// TwinCAT 3 PLC project PLC_FIS
// ProgramVersion: 3.1.4024.12
// libraries:
//   Tc2_Standard, * (Beckhoff Automation GmbH)
//   Tc2_System, * (Beckhoff Automation GmbH)
//   Tc3_Module, * (Beckhoff Automation GmbH)
// project tree:
//   DUTs/ eAndMethod.TcDUT, eDeffuzyMethod.TcDUT (not stored), eOrMethod.TcDUT (not stored), eTest.TcDUT, MAMFIS.TcDUT, FIS_RULES.TcDUT, FIS_VAR.TcDUT, FIS_VAR_1.TcDUT (not stored), MF_INDEX.TcDUT, MF_SHAPE.TcDUT, MEMBERSHIP_FUNCTION.TcDUT (not stored)
//   GVLs/ gvlFIS_Constants.TcGVL
//   Old/ fbFuzzyAnd.TcPOU, fCentroidOld.TcPOU, fIntegrateMf.TcPOU, fIntExtFun.TcPOU, fis_cfc.TcPOU, fLinInterpol.TcPOU, LINEAR_LUT.TcPOU, LINEAR_LUT_old.TcPOU, mySumFb.TcPOU, testReferenceToFB.TcPOU
//   OOP/ FB_FIS_oop.TcPOU, FuzzyInferenceSystem.TcIO, OOP_MAIN.TcPOU
//   / PlcTask.TcTTO (not stored)
//   POP/Deffuzzification/ fCentroid.TcPOU (not stored)
//   POP/ FB_AGGREGATION.TcPOU (not stored), FB_IMPLICATION.TcPOU (not stored), FIS_pgr.TcPOU, MAIN.TcPOU
//   POP/Fuzzification/ fMembershipDegree.TcPOU, fMembershipDegreeArray.TcPOU
//   POP/Fuzzification/Membership Functions/ MF_Gaussian.TcPOU, MF_L.TcPOU, MF_R.TcPOU, MF_S.TcPOU (not stored), MF_Sigmoidal.TcPOU, MF_Singleton.TcPOU, MF_Trapezoidal.TcPOU (not stored), MF_Triangular.TcPOU, MF_Z.TcPOU
//   POP/FuzzyOperations/ fuzzyset.TcPOU, FuzzyAND_array.TcPOU (not stored), fuzzyAND.TcPOU, FuzzyNOT.TcPOU, FuzzyOR_array.TcPOU (not stored), FuzzyOR.TcPOU
//   POP/FuzzyOperations/T-Norms/ TN_min.TcPOU (not stored), TN_prod.TcPOU
//   POP/Test/ Test_fbFis.TcPOU (not stored)
//   POP/_FuzzyInferenceSystem/ FB_FIS_MAMDANI.TcPOU

// ---- DUTs/eAndMethod.TcDUT
//{attribute 'qualified_only'}
{attribute 'strict'}
TYPE eAndMethod :
(
	Minimum,
	Product
);
END_TYPE

// ---- DUTs/eTest.TcDUT
{attribute 'qualified_only'}
{attribute 'strict'}
TYPE eTest :
(
	enum_member := 0
);
END_TYPE

// ---- DUTs/MAMFIS.TcDUT
TYPE MAMFIS :
	STRUCT
		Name:STRING;
		Rules:ARRAY[1..NumOfFisRules]OF FIS_RULES;
		AndMethod:eAndMethod;
		OrMethod:eOrMethod;
		ImplicationMethod:eAndMethod; 
		AggregationMethod:eOrMethod;
		DefuzzificationMethod:eDeffuzyMethod;
		Inputs:ARRAY[1..NumOfFISInputs]OF FIS_VAR;
		MD:ARRAY[1..NumOfFISInputs,1..MFmax]OF REAL;//MD
		Outputs:ARRAY[1..NumOfFISOutputs]OF FIS_VAR;
	END_STRUCT
END_TYPE

// ---- DUTs/FIS_RULES.TcDUT
TYPE FIS_RULES :
STRUCT
	Antecedent: REAL;
	Consequents:ARRAY[1..NumOfFISOutputs]OF MF_INDEX;
END_STRUCT
END_TYPE

// ---- DUTs/FIS_VAR.TcDUT
TYPE FIS_VAR :
STRUCT
	CrispValue:REAL;
	Name:STRING;
	Range:ARRAY[1..2] OF REAL;
	NumberOfMF:INT;
	MF:ARRAY [1..MFmax]OF MEMBERSHIP_FUNCTION;//MF

END_STRUCT
END_TYPE

// ---- DUTs/MF_INDEX.TcDUT
TYPE
	MF_INDEX : INT;
END_TYPE

// ---- DUTs/MF_SHAPE.TcDUT
{attribute 'qualified_only'}
{attribute 'strict'}
TYPE MF_SHAPE :
(
	Gaussian,
	Lshaped,
	Rshaped,
	Sshaped,
	Sigmoidal,
	Singleton,
	Trapeziodal,
	Triangular,
	Zshaped
);
END_TYPE

// ---- GVLs/gvlFIS_Constants.TcGVL
{attribute 'global'}
VAR_GLOBAL CONSTANT
	NumOfFISInputs:INT :=	2;
	NumOfFISOutputs:INT := 	1;
	MFmax:INT := 			3;//maximum of MF per variable
	NumOfFisRules:INT := 	3;
	
	//inputs
	 	Error:INT:=1;
	 	Speed:INT:=2;
		
	//outputs
	 	power:INT:=1;
		
	//INPUT MEMBERSHIP FUNCTIONS
		None:INT := 	 1;
		Little:INT := 	 2;	
		Big:INT := 	 3;		
		//Negative:INT := 1;
		//Null:INT :=	 2;
		//Positive:INT := 3;
		
	//OUTPUT MEMBERSHIP FUNCTIONS
		Low:INT := 1;
		Medium:INT :=	 2;
		High:INT := 3;
END_VAR

// ---- OOP/FuzzyInferenceSystem.TcIO
INTERFACE FuzzyInferenceSystem

METHOD Defuzzification :REAL;
VAR_INPUT
END_VAR
END_METHOD

METHOD Fuzzyfication 
VAR_INPUT
END_VAR
END_METHOD

END_INTERFACE

// ---- Old/fbFuzzyAnd.TcPOU
FUNCTION_BLOCK fbFuzzyAnd
VAR_INPUT
END_VAR
VAR_OUTPUT
END_VAR
VAR
END_VAR

END_FUNCTION_BLOCK

// ---- Old/fCentroidOld.TcPOU
FUNCTION fCentroidOld : REAL
VAR_INPUT
	Range:ARRAY[1..2] OF REAL;
	MF:MEMBERSHIP_FUNCTION;
	Resolution:DINT;
END_VAR
VAR
	i:DINT;
	Xi,MDi,Step:REAL;
	Dividend:REAL:=0;//sum(MD(Xi))
 	Divisor:REAL:=0;//sum(Xi*MD(Xi))
END_VAR

(*
centroid=   sum(MD(Xi))  dividend
		  ==============
		  sum(Xi*MD(Xi)) divisor
*)
Step:=Range[2]-Range[1];
IF Resolution<>0 THEN
	FOR i := 1 TO resolution DO
		Xi := DINT_TO_REAL(i)*Step/Resolution;
		MDi := fMembershipDegree(Xi,MF);
		Dividend := Dividend + MDi;
		Divisor :=Divisor+(Mdi*Xi);
	END_FOR
	IF Divisor<>0 THEN
		fCentroidOld := Dividend/Divisor;
	ELSE
		fCentroidOld:=0;
	END_IF
ELSE fCentroidOld:=666;	
END_IF

END_FUNCTION

// ---- POP/Fuzzification/fMembershipDegree.TcPOU
FUNCTION fMembershipDegree : real
VAR_INPUT
	CrispInput: REAL;
	MF:MEMBERSHIP_FUNCTION;
END_VAR

VAR_OUTPUT
	error: BOOL;
END_VAR

CASE MF.Shape OF
	MF_SHAPE.Gaussian://********
		fMembershipDegree:=
			MF_Gaussian(
				x:= CrispInput,
				c:= MF.Points[1],
				d:= MF.Points[2],
				Error=>error);
	MF_SHAPE.Lshaped://********
		fMembershipDegree:=
			MF_L(
				x:= CrispInput,
				a:= MF.Points[1],
				b:= MF.Points[2],
				Error=>error);

	MF_SHAPE.rshaped://********
		fMembershipDegree:=
			MF_R(
				x:= CrispInput,
				c:= MF.Points[1],
				d:= MF.Points[2],
				Error=>error);
	
	MF_SHAPE.Sshaped://********
		fMembershipDegree:=
			MF_S(
				x:= CrispInput,
				a:= MF.Points[1],
				b:= MF.Points[2],
				Error=>error);

	MF_SHAPE.Sigmoidal://********
		fMembershipDegree:=
			MF_Gaussian(
				x:= CrispInput,
				d:= MF.Points[1],
				c:= MF.Points[2],
				Error=>error);
							
	MF_SHAPE.Singleton://********
		fMembershipDegree:=
			MF_Singleton(
				x:= CrispInput,
				a:= MF.Points[1]);
				
	MF_SHAPE.Trapeziodal://********
		fMembershipDegree:=
			MF_Trapezoidal(
				x:= CrispInput,
				a:= MF.Points[1],
				b:= MF.Points[2],
				c:= MF.Points[3],
				d:= MF.Points[3],
				Error=>error);
	
	MF_SHAPE.Triangular://********	
		fMembershipDegree:=
			MF_Triangular(
				x:= CrispInput,
				a:= MF.Points[1],
				m:= MF.Points[2],
				b:= MF.Points[3],
				error=>error);
				
	MF_SHAPE.Zshaped://********
		fMembershipDegree:=
			MF_R(
				x:= CrispInput,
				c:= MF.Points[1],
				d:= MF.Points[2],
				Error=>error);
	ELSE
		error:=TRUE;
	END_CASE;

END_FUNCTION

// ---- POP/Fuzzification/Membership Functions/MF_Gaussian.TcPOU
FUNCTION MF_Gaussian : real
VAR_INPUT
	x,d,c:REAL;(*Membership function parameters,
specified as the vector [d c], where σ is the 
standard deviation AND c is the mean.*)
END_VAR
VAR_OUTPUT
	Error:BOOL;
END_VAR

IF NOT(d=0) THEN
	MF_Gaussian := LREAL_TO_REAL(EXP(-EXPT((x-c),2)/EXPT(2*d,2)));
ELSE
	Error:=TRUE;
END_IF

END_FUNCTION

// ---- POP/Fuzzification/Membership Functions/MF_L.TcPOU
FUNCTION MF_L : real
VAR_INPUT
	x,a,b:REAL;(*a defines the foot of the membership function, AND b defines its shoulder.*)

END_VAR
VAR_OUTPUT
	Error:BOOL;
END_VAR

IF NOT(a=b) AND (a<b) THEN
	IF x<a THEN
		MF_L:=0;
	ELSIF a<=x AND x<=b THEN
		MF_L:=(x-a)/(b-a);
	ELSIF  x>b THEN
		MF_L:=1;
	END_IF
ELSE
	Error:=TRUE;		
END_IF

END_FUNCTION

// ---- POP/Fuzzification/Membership Functions/MF_R.TcPOU
 FUNCTION MF_R : real
VAR_INPUT
	x,d,c:REAL;(*a defines the foot of the membership function, AND b defines its shoulder.*)

END_VAR
VAR_OUTPUT
	Error:BOOL;
END_VAR

IF NOT(c=d) AND (c<d) THEN
	IF x>d THEN
		MF_R:=0;
	ELSIF c<=x AND x<=d THEN
		MF_R:=(d-x)/(d-c);
	ELSIF  x<c THEN
		MF_R:=1;
	END_IF
ELSE
	Error:=TRUE;		
END_IF

END_FUNCTION

// ---- POP/Fuzzification/Membership Functions/MF_Singleton.TcPOU
FUNCTION MF_Singleton : real
VAR_INPUT
	x,a:REAL;
END_VAR
VAR
END_VAR

IF x=a then
	MF_Singleton:=1;
ELSE
	MF_Singleton:=0;
END_IF

END_FUNCTION

// ---- POP/Fuzzification/Membership Functions/MF_Triangular.TcPOU
FUNCTION MF_Triangular : real
VAR_INPUT
	x,a,m,b:REAL;
END_VAR
VAR_OUTPUT
	error: BOOL;
END_VAR

// a < m < b
IF (a<m) AND (m<b) THEN
	IF x<=a OR x>=b THEN
		MF_Triangular:=0;
	ELSIF a<x AND x<m THEN
		MF_Triangular:=(x-a)/(m-a);
	ELSIF m<=x AND x<=b THEN
		MF_Triangular:=(b-x)/(b-m);
	END_IF
ELSE
	error:=TRUE;		
END_IF

END_FUNCTION

// ---- Old/fIntegrateMf.TcPOU
FUNCTION fIntegrateMf : real
VAR_INPUT
	resolution:DINT;//number of integration rectangles
	Range:ARRAY[1..2] OF REAL;
	refFbFuzzySet: REFERENCE TO FB_FUZZY_SET;//MF:MEMBERSHIP_FUNCTION;
END_VAR
VAR
	i:DINT;
	Xi,MDi:REAL;
	IntegrationStep: REAL;
END_VAR

IF Resolution<>0 THEN
IntegrationStep:=(Range[2]-Range[1])/DINT_TO_REAL(Resolution);
	FOR i := 1 TO resolution DO
		xi:=DINT_TO_REAL(i);//Xi := DINT_TO_REAL(i)*IntegrationStep;
		refFbFuzzySet(X:=Xi);
		MDi := refFbFuzzySet.FSValue;
		fIntegrateMf := fIntegrateMf +MDi;// MDi*IntegrationStep;
	END_FOR
END_IF

END_FUNCTION

// ---- Old/fIntExtFun.TcPOU
FUNCTION fIntExtFun : real
VAR_INPUT
	Range:ARRAY[1..2] OF REAL;
	resolution:DINT;//number of integration rectangles
END_VAR
VAR
	i:DINT;
	Xi,MDi:REAL;
	IntegrationStep: REAL;
END_VAR

IF Resolution<>0 THEN
	//calcular el paso de integracion
	IntegrationStep:=(Range[2]-Range[1])/DINT_TO_REAL(Resolution);
	
	FOR i := 1 TO resolution DO
		Xi := DINT_TO_REAL(i)*IntegrationStep;//paso de integracion actual
		MDi :=Extfun(Xi) ;//llamada a la funcion abstracta
		fIntegrateMf := fIntExtFun + MDi*IntegrationStep;
	END_FOR
END_IF

END_FUNCTION

// ---- Old/fis_cfc.TcPOU
FUNCTION_BLOCK fis_cfc
VAR_INPUT
	crispinput1:real;
END_VAR

VAR
mymf:MEMBERSHIP_FUNCTION:=(mymf.Name:='error',Points:=[1,2,3,4,5]);
END_VAR

VAR_OUTPUT
END_VAR
VAR
	FB_FIS_0: fb_fis;
END_VAR
VAR // added by the converter: edge detectors and wires of the graphical bodies
    _w1, _w2, _w3 : BOOL;
END_VAR

FB_FIS_0(); // fb_fis
fMembershipDegree();
(* _w1 OR _w2 OR _w3; result not used *)
fMembershipDegree(MF := CrispInput1, error => _w3);
fMembershipDegree(CrispInput := CrispInput1, error => _w2);
fMembershipDegree(CrispInput := CrispInput1, MF := mymf, error => _w1);

END_FUNCTION_BLOCK

// ---- Old/fLinInterpol.TcPOU
FUNCTION fLinInterpol : real
VAR_INPUT
	InputValue,Xmin,Xmax,Ymin,Ymax:REAL;
END_VAR
VAR
	b,a:REAL;
END_VAR

//y=a+bx
b:= YMin+InputValue*((Xmax-Xmin)/(Ymax-Ymin));
a:= Ymin-b*xmin;
fLinInterpol:=a+b*InputValue;

END_FUNCTION

// ---- Old/LINEAR_LUT.TcPOU
FUNCTION LINEAR_LUT : REAL
VAR_INPUT
	rInput:REAL;
END_VAR

VAR_IN_OUT	
	XCol,YCol: ARRAY[*] OF REAL;
END_VAR

VAR
	i,Array1st,ArrayLast: DINT;
	XIncrement:REAL;
END_VAR

Array1st:= LOWER_BOUND(XCol,1);
ArrayLast:= UPPER_BOUND(XCol,1);

IF rInput<= Xcol[Array1st] THEN
	LINEAR_LUT:=YCol[Array1st];
ELSIF rInput>= XCol[ArrayLast] THEN
	LINEAR_LUT:=YCol[ArrayLast];
ELSE
	FOR i:=Array1st TO ArrayLast-1 DO
		IF rInput >= XCol[i] THEN
			XIncrement:= XCol[i+1]-XCol[i];
			IF XIncrement=0 THEN
				LINEAR_LUT:=YCol[i];
			ELSE	
				LINEAR_LUT:=YCol[i]+(rInput-Xcol[i])*(YCol[i+1]-YCol[i])/XIncrement;
				RETURN;
			END_IF;
		END_IF
	END_FOR
END_IF

END_FUNCTION

// ---- Old/LINEAR_LUT_old.TcPOU
FUNCTION LINEAR_LUT_old : REAL
VAR_INPUT
	rInput:REAL;
	InputCol: ARRAY[0..10] OF REAL;
	OutputCol: ARRAY[0..10] OF REAL;
END_VAR
VAR
	i: INT;
END_VAR
VAR CONSTANT
	Array1st:INT:=0;
	ArrayLast:INT:=10;
END_VAR

IF rInput<= InputCol[Array1st] THEN
	LINEAR_LUT_old:=OutputCol[Array1st];
ELSIF rInput>= InputCol[ArrayLast] THEN
	LINEAR_LUT_old:=OutputCol[ArrayLast];
ELSE
	FOR i:=Array1st TO ArrayLast-1 DO
		IF rInput >= InputCol[i] THEN
			LINEAR_LUT_old:=OutputCol[i]+(rInput-inputcol[i])*(OutputCol[i+1]-OutputCol[i])/(InputCol[i+1]-InputCol[i]);
			RETURN;
		END_IF
	END_FOR
END_IF

END_FUNCTION

// ---- Old/mySumFb.TcPOU
FUNCTION_BLOCK mySumFb
VAR_INPUT
	sum1,sum2:REAL;
END_VAR
VAR_OUTPUT
	result:real;
END_VAR
VAR
END_VAR

result := sum1+sum2;

END_FUNCTION_BLOCK

// ---- Old/testReferenceToFB.TcPOU
FUNCTION testReferenceToFB :ARRAY [1..2]OF  REAL
VAR_INPUT
	RefSum: REFERENCE TO mySumFb;
	PointerSum: POINTER TO mySumFb;
	sum2:REAL;
END_VAR
VAR
		MyFb_p_Sum:mySumFb;
END_VAR

MyFb_p_Sum := PointerSum^;

RefSum.sum2:=sum2;
testReferenceToFB[1]:=MyFb_p_Sum.result;
testReferenceToFB[2]:=RefSum.result;

END_FUNCTION

// ---- OOP/FB_FIS_oop.TcPOU
FUNCTION_BLOCK FB_FIS_oop IMPLEMENTS FuzzyInferenceSystem
VAR_INPUT
END_VAR
VAR_OUTPUT
END_VAR
VAR
END_VAR

END_FUNCTION_BLOCK

// ---- OOP/OOP_MAIN.TcPOU
PROGRAM OOP_MAIN
VAR
	FuzzyLogicController:FB_FIS_oop;
	
END_VAR

END_PROGRAM

// ---- POP/FIS_pgr.TcPOU
PROGRAM FIS_pgr
VAR
	CrispInputsSimulation: ARRAY[1..NumOfFISInputs] OF REAL;
	Inputs: ARRAY[1..NumOfFISInputs] OF FIS_VAR;
	MD:ARRAY[1..NumOfFISInputs,1..MFmax]OF REAL;//MD
	Outputs: ARRAY[1..NumOfFISOutputs] OF FIS_VAR;
	Rules:ARRAY [1..NumOfFisRules] OF FIS_RULES;
	i,j: DINT;	
	fbAggregation:FB_AGGREGATION;
END_VAR

//FUZZY INFERENCE SYSTEM 
//======================================================

//INPUTS DEFINITION
	//input1=ERROR(command-feedback)
		Inputs[1].CrispValue:=	CrispInputsSimulation[1];
		Inputs[1].Name  :=  	'TempError';
		Inputs[1].Range[1] :=  	0;
		Inputs[1].Range[2] := 	70;
		Inputs[1].NumberOfMF := 3;
		
		Inputs[1].MF[1].Name := 	'none';
		Inputs[1].MF[1].Shape := 	MF_SHAPE.Rshaped;
		Inputs[1].MF[1].Points[1] := 0;
		Inputs[1].MF[1].Points[2] := 10;
		
		Inputs[1].MF[2].Name := 	'litle';
		Inputs[1].MF[2].Shape := 	MF_SHAPE.Triangular;
		Inputs[1].MF[2].Points[1] := 5;
		Inputs[1].MF[2].Points[2] := 20;
		Inputs[1].MF[2].Points[3] := 40;
		
		Inputs[1].MF[3].Name := 	'big';                                                                                 
		Inputs[1].MF[3].Shape := 	MF_SHAPE.Lshaped;
		Inputs[1].MF[3].Points[1] := 20;
		Inputs[1].MF[3].Points[2] := 60;	
										 
	//input2=differror
		Inputs[2].CrispValue:=	CrispInputsSimulation[2];
		Inputs[2].Name := 		'speed';
		Inputs[2].Range[1] :=  	0;
		Inputs[2].Range[2] := 	20;
		Inputs[2].NumberOfMF := 3;
		
		Inputs[2].MF[1].Name := 	'null';
		Inputs[2].MF[1].Shape := 	MF_SHAPE.Rshaped;
		Inputs[2].MF[1].Points[1] := 0;
		Inputs[2].MF[1].Points[2] := 2;
		
		Inputs[2].MF[2].Name := 	'litlle';
		Inputs[2].MF[2].Shape := 	MF_SHAPE.Triangular;
		Inputs[2].MF[2].Points[1] := 0;
		Inputs[2].MF[2].Points[2] := 5;
		Inputs[2].MF[2].Points[3] := 10;
		
		Inputs[2].MF[3].Name := 	'Big';
		Inputs[2].MF[3].Shape := 	MF_SHAPE.Lshaped;
		Inputs[2].MF[3].Points[1] := 8;
		Inputs[2].MF[3].Points[2] := 15;
//======================================================

//FUZZY OUTPUTS DEFINITION 
	Outputs[1].Name  :=  		'Power';
	Outputs[1].Range[1] :=  	0;
	Outputs[1].Range[2] :=		120;
	Outputs[1].NumberOfMF := 	3;
	
	Outputs[1].MF[1].Name := 	'Low';
	Outputs[1].MF[1].Shape := 	MF_SHAPE.Rshaped;
	Outputs[1].MF[1].Points[1] := 0;
	Outputs[1].MF[1].Points[2] := 30 ;

	
	Outputs[1].MF[2].Name := 	'Medium';
	Outputs[1].MF[2].Shape := 	MF_SHAPE.Triangular;
	Outputs[1].MF[2].Points[1] := 20;
	Outputs[1].MF[2].Points[2] := 40;
	Outputs[1].MF[2].Points[3] := 60;
	
	Outputs[1].MF[3].Name := 	'High';
	Outputs[1].MF[3].Shape := 	MF_SHAPE.Lshaped;
	Outputs[1].MF[3].Points[1] := 50;
	Outputs[1].MF[3].Points[2] := 100;
//======================================================

//Fuzzufication inteface				
	//Membership degrees calculation 
	//---is interesting calculate directlu con antecedents calculation?
	FOR i:=1 TO NumOfFISInputs DO
		FOR j:=1 TO inputs[i].NumberOfMF DO
			MD[i,j]:= 
				fMembershipDegree(
					CrispInput := Inputs[i].CrispValue,
					MF:= Inputs[i].MF[j]);
		END_FOR	 
	END_FOR
//======================================================

//FUZZY_rules
	//Rules[1].Antecedent := fuzzyAND(Minimum,MD[error,none],MD[speed,None]);
	Rules[1].Antecedent := MD[error,none];
	Rules[1].Consequents[power] := low;
	
	//Rules[2].Antecedent:= FuzzyAND(Minimum,MD[error,little],MD[speed,little]);
	Rules[2].Antecedent:=MD[error,little];
	Rules[2].Consequents[power] := medium;
	
	//Rules[3].Antecedent:= fuzzyAND(Minimum,MD[error,big],MD[speed,big]);
	Rules[3].Antecedent:= MD[error,big];
	Rules[3].Consequents[power] := High;
//======================================================

	
//Aggregation
fbAggregation.Myrules:=Rules;
fbAggregation.MyFISoutputs:=Outputs;
//Deffuzification
Outputs[1].CrispValue:=fCentroid(100,Outputs[1].Range,fbAggregation);

END_PROGRAM

// ---- POP/Fuzzification/fMembershipDegreeArray.TcPOU
FUNCTION fMembershipDegreeArray : REAL;
VAR
	i,j:DINT;
END_VAR
VAR_IN_OUT
	FisVariables:ARRAY[*]OF FIS_VAR;
	MD : ARRAY[*  , *  ] OF REAL;
//MD:ARRAY[*]OF ARRAY[*] OF REAL;
END_VAR
VAR_OUTPUT
	error: BOOL;
END_VAR

FOR i:=LOWER_BOUND(FisVariables,1) TO UPPER_BOUND(FisVariables,1) DO
	FOR j:=1 TO FisVariables[I].NumberOfMF DO
		MD[i,j]:= 
			fMembershipDegree(
				CrispInput := FisVariables[i].CrispValue,
				MD[i,j] := FisVariables[i].MF[j]);
	END_FOR	
END_FOR

END_FUNCTION

// ---- POP/Fuzzification/Membership Functions/MF_Sigmoidal.TcPOU
FUNCTION MF_Sigmoidal : REAL
VAR_INPUT
	x,a,c:REAL;
END_VAR
VAR
	divisor: REAL;
END_VAR

VAR_OUTPUT
	error: BOOL;
END_VAR

divisor:=1+LREAL_TO_REAL(EXP(-a*(x-c)));
IF divisor<>0 THEN	
	MF_Sigmoidal:=1/divisor;
	ELSE error:=TRUE;
END_IF;

END_FUNCTION

// ---- POP/Fuzzification/Membership Functions/MF_Z.TcPOU
FUNCTION MF_Z : real
VAR_INPUT
	x,a,b:REAL;(*a defines the foot of the membership function, AND b defines its shoulder.*)

END_VAR
VAR_OUTPUT
	Error:BOOL;
END_VAR

IF NOT(b=a) THEN
	IF x<=a THEN
		MF_Z := 0;
	ELSIF a<=x AND x<=(a+b)/2 THEN
		MF_Z := 1 - 2*EXPT(((x-a)/(b-a)),2);
	ELSIF (a+b)/2<=x AND x<=b THEN
		MF_Z := 2*EXPT(((x-B)/(b-a)),2);
	ELSIF b<=x THEN
		MF_Z := 1;
	END_IF
ELSE
	Error:=TRUE;
END_IF

END_FUNCTION

// ---- POP/FuzzyOperations/fuzzyset.TcPOU
FUNCTION fuzzyset : ARRAY [1..100]OF REAL;
VAR_INPUT
	antecedent:REAL;
END_VAR
VAR_IN_OUT
	outputs: ARRAY[*] OF FIS_VAR;
END_VAR

VAR
	i,j,Array1st,ArrayLast,NumOfInputs: DINT;
END_VAR

Array1st:= LOWER_BOUND(Inputs,1);
ArrayLast:= UPPER_BOUND(Inputs,1);
//calcular la impicaxionFOR i:=Array1st TO ArrayLast DO
//CASE MF.Shape OF
//	mf_shape.Singleton://
//;//transparente
//	mf_shape.Triangular://
//;//	sale un trpaecio
//END_CASE
//
FOR i:=1 TO i=100 DO
fuzzyAND(minimum,antecedent,fMembershipDegree())

//IF haciendo el MAX de las funciones de mf implicadas

END_FUNCTION

// ---- POP/FuzzyOperations/fuzzyAND.TcPOU
FUNCTION fuzzyAND : REAL
VAR_INPUT
	ANDmethod:eAndMethod;
	in1,in2:REAL;
END_VAR

CASE ANDmethod OF
	eAndMethod.Minimum://***********
		fuzzyAND := MIN(in1,in2);
	eAndMethod.Product://***********
		fuzzyAND := in1*in2;
END_CASE

END_FUNCTION

// ---- POP/FuzzyOperations/FuzzyNOT.TcPOU
FUNCTION FuzzyNOT : REAL
VAR_INPUT
	MD:REAL;//MEMBERSHIP DEGREE
END_VAR
VAR
END_VAR

FuzzyNOT:=1-MD;

END_FUNCTION

// ---- POP/FuzzyOperations/FuzzyOR.TcPOU
FUNCTION FuzzyOR : real
VAR_INPUT
	ORmethod:eORMethod;
	in1,in2:REAL;
END_VAR

CASE ORmethod OF
	Maximum:
		FuzzyOR:=MAX(in1,in2);
END_CASE

END_FUNCTION

// ---- POP/FuzzyOperations/T-Norms/TN_prod.TcPOU
FUNCTION TN_prod : real
VAR
	i:DINT;
END_VAR
VAR_IN_OUT
	Inputs: ARRAY[*] OF REAL;
END_VAR

TN_prod:=1;
FOR i:=LOWER_BOUND(Inputs,1) TO UPPER_BOUND(Inputs,1) DO
	TN_prod:=TN_prod*inputs[i];
END_FOR

END_FUNCTION

// ---- POP/MAIN.TcPOU
PROGRAM MAIN
VAR
END_VAR

FIS_pgr();

Test_fbFis();

END_PROGRAM

// ---- POP/_FuzzyInferenceSystem/FB_FIS_MAMDANI.TcPOU
FUNCTION_BLOCK FB_FIS_MAMDANI
VAR_IN_OUT
	FIS:MAMFIS;
END_VAR
VAR
	i,j: DINT;	
	fbAggregation:FB_AGGREGATION;
END_VAR

//Fuzzufication inteface				
	//Membership degrees calculation 
	FOR i:=1 TO NumOfFISInputs DO
		FOR j:=1 TO FIS.inputs[i].NumberOfMF DO
			FIS.MD[i,j]:= 
				fMembershipDegree(
					CrispInput := FIS.Inputs[i].CrispValue,
					MF:= FIS.Inputs[i].MF[j]);
		END_FOR	 
	END_FOR
//Implication: ImplicationFB is called By FBAggregation

//Aggregation FBis called by Deffuzification function
	fbAggregation.Myrules:=FIS.Rules;
	fbAggregation.MyFISoutputs:=FIS.Outputs;
//Deffuzification
	FIS.Outputs[1].CrispValue:=fCentroid(100,FIS.Outputs[1].Range,fbAggregation);

END_FUNCTION_BLOCK
